// SIMATIC S7-200 project (STEP 7-Micro/WIN), CPU 221 REL 01.10

ORGANIZATION_BLOCK 主:OB1
TITLE=程序注释
// PLC通过PID算法自动调节加热器的输出功率，使反应釜温度趋于稳定，以满足化学反应需求。系统在PLC首次上电时，检测到首次扫描标志为1，调用子程序，设置PID循环定点为0.615（对应温度范围的61.5%）、PID循环增益为2.0、PID循环采样时间为0.1秒、PID积分时间为4.0分钟、PID微分时间为0.0（不启用微分控制）。同时，系统将定时器间隔配置为10毫秒，并附加PID执行中断，保证PID控制以10毫秒周期执行——只有这些参数正确初始化，系统才能正常运行。
// 在每个10毫秒周期内，PID执行中断启动，PLC读取温度传感器输入，将其转换为PID过程变量作为当前温度测量值。当自动模式开关为1时，系统计算PID输出并调整加热控制输出，以实现加热强度的自动调节。为确保温度数据实时可见，常开标志驱动下，系统将PID过程变量和PID循环定点转换为检测温度显示值和设定温度显示值，并通过数据传输标志发送至PC机，以实现实时监控。
// 若温度超限，主程序监控PID过程变量是否大于等于PID循环定点，并将加热控制输出设为16000以降低温度。超温时，系统需避免加热控制输出在下一周期被意外调整，以确保温度安全。加热器开关阈值用于控制加热器开关的状态，根据PID输出调整加热强度。此外，加热器开关阈值控制加热器开关：大于10000时关闭，小于6000时开启——在6000至10000之间若加热器开关保持开启，可能导致温度持续上升超出PID循环定点。当温度超出设定范围时，系统可关闭加热器以维持温度稳定。
BEGIN
Network 1 // 设置通讯方式，调用传送PID参数子程序，启动TD200使能位。
//  
// 网络注释
//  
// 
LD     SM0.1
MOVB   9, SMB30
MOVB   0, SMB130
CALL   SBR_0:SBR0
MOVB   16#80, VB12
MOVB   0, MB0
?000
Network 2 // 传送向PC机发送的数据表。
// 
// 
LD     SM0.0
MOVB   4, VB199
MOVW   VW56, VW200
MOVW   VW76, VW202
Network 3 // 向PC机发送数据。
// 
// 
LD     SM0.5
EU
XMT    VB199, 0
Network 4 // 超过额温度限制输出。
// 
// 
LDD>=  VD100, VD104
MOVW   +16000, AQW0
Network 5 // 温控时间的计数器（单位为秒）。
// 
// 
LD     SM0.5
LD     SM0.1
CTU    C0, +0
Network 6 // 计算检测的温度参数，传送到VW556。设定的温度参数传送到VW576。
// 
// 
LD     SM0.0
MOVR   VD100, AC0
*R     32000.0, AC0
ROUND  AC0, AC0
DTI    AC0, VW556
MOVR   VD104, AC0
*R     32000.0, AC0
ROUND  AC0, AC0
DTI    AC0, VW576
Network 7 // 检测的温度值送VW56，设定温度值送VW76。
// 
// 
LD     SM0.0
-I     +6552, VW556
MOVW   VW556, VW56
/I     +131, VW56
-I     +6552, VW576
MOVW   VW576, VW76
/I     +131, VW76
END_ORGANIZATION_BLOCK

SUBROUTINE_BLOCK SBR_0:SBR0
TITLE= 
// 子程序注释
// 按 F1 获得帮助及举例程序
//  
// 
BEGIN
Network 1 // 传送PID参数。
//  
// 网络注释
//  
// 
LD     SM0.0
MOVR   0.615, VD104
MOVR   2.0, VD112
MOVR   0.1, VD116
MOVR   4.0, VD120
MOVR   0.0, VD124
MOVB   10, SMB34
ATCH   INT_0:INT0, 10
ENI
END_SUBROUTINE_BLOCK

INTERRUPT_BLOCK INT_0:INT0
TITLE= 
// 中断程序注释
// 按 F1 获得帮助及举例程序
//  
// 
BEGIN
Network 1 // 检测温度参数送PID参数表。
//  
// 网络注释
//  
// 
LD     SM0.5
EU
MOVW   AIW0, VW402
DTR    VD400, VD404
MOVR   VD404, VD408
/R     32000.0, VD408
MOVR   VD408, VD100
Network 2 // I0.0=1,计算PID输出。
// 
// 
LD     I0.0
PID    VB100, 0
Network 3 // 根据PID输出通过D/A模块控制调压模块（DC 0-5V）。
// 
// 
LD     SM0.0
MOVR   VD108, AC0
*R     16000.0, AC0
ROUND  AC0, AC0
DTI    AC0, VW310
MOVW   +16000, VW304
-I     VW310, VW304
MOVW   VW304, AQW0
Network 4 // ****用Q0.0控制交流220V的输出。
// 
// 
LD     SM0.0
LPS
AW>    VW304, +10000
R      Q0.0, 1
LPP
AW<    VW304, +6000
S      Q0.0, 1
END_INTERRUPT_BLOCK
